INTERFACE ITF_Device EXTENDS ITF_BASE

PROPERTY Homed : BOOL
GET
END_GET
SET
END_SET
END_PROPERTY

METHOD mAbort : E_CmdState
VAR_INPUT
	I_bExecute : BOOL;
END_VAR
END_METHOD

METHOD mAutomatic : E_CmdState
VAR_INPUT
	I_bExecute : BOOL;
END_VAR
END_METHOD

METHOD mDone : E_CmdState
VAR_INPUT
END_VAR
END_METHOD

METHOD mHold : E_CmdState
VAR_INPUT
	I_bExecute : BOOL;
END_VAR
END_METHOD

METHOD mHome : E_CmdState
VAR_INPUT
	I_bExecute : BOOL;
END_VAR
END_METHOD

PROPERTY Mode : E_Mode
GET
END_GET
SET
END_SET
END_PROPERTY

METHOD mRelease : E_CmdState
VAR_INPUT
	I_bExecute : BOOL;
END_VAR
END_METHOD

METHOD mSequence : E_CmdState
VAR_INPUT
	I_bExecute : BOOL;
END_VAR
END_METHOD

METHOD mService : E_CmdState
VAR_INPUT
	I_bExecute : BOOL;
END_VAR
END_METHOD

METHOD mStop : E_CmdState
VAR_INPUT
	I_bExecute : BOOL;
END_VAR
END_METHOD

PROPERTY Ready : BOOL
GET
END_GET
SET
END_SET
END_PROPERTY

PROPERTY SequenceBusy : BOOL
GET
END_GET
SET
END_SET
END_PROPERTY

PROPERTY SequenceDone : BOOL
GET
END_GET
SET
END_SET
END_PROPERTY

END_INTERFACE

(* stored: Version 1.1.0.1, ProductVersion 3.1.4026.18
   Itf ITF_Device: Id {7c7c0ada-9da2-4ea4-a6eb-5bdbbf502dd6}
   Folder 01 Properties: Id {cc599803-8df0-4524-b56e-e6f8332deeb0}
   Folder 02 Methode: Id {8d03e7f7-1295-4a10-8500-54223f6c93df}
   Property Homed: Id {e0b0dbb4-f26b-41da-9728-17a21e3e50b5}
   Get Get: Id {b29716a5-bb80-4dae-9f4b-48cd3af13c02}
   Set Set: Id {c173668d-1e20-490e-b2a6-a314d734dc62}
   Method mAbort: Id {c49357ee-7419-4b69-b3cb-4341d2ee13d7}
   Method mAutomatic: Id {2d6cc853-f349-4892-b830-c8d902fec512}
   Method mDone: Id {ab0168ac-f476-4285-a122-68c9646e188c}
   Method mHold: Id {731bcd95-814c-4609-aa5e-a6712b35be37}
   Method mHome: Id {8c5e9607-f090-4f86-b53e-de4094b3fc51}
   Property Mode: Id {b4148d7b-1cf4-4690-8b11-f60ccf8fdb97}
   Get Get: Id {1764c7ca-5320-4c72-952b-b11de84e4a86}
   Set Set: Id {84b839d5-3e71-4766-9ef6-014419011dfe}
   Method mRelease: Id {39840917-54ed-488a-8e37-97e1ca73b28a}
   Method mSequence: Id {2de450d3-e14b-44df-ad83-42812f65ff1e}
   Method mService: Id {77e7e75c-3f71-4063-a921-5cc7e456b4a1}
   Method mStop: Id {dcef2cbd-175d-4efc-8e1c-1281a72f37b3}
   Property Ready: Id {47c16123-6529-4896-a7e2-12f8732a490d}
   Get Get: Id {0ffcaf96-efe5-4f3a-a02e-5895995aeb20}
   Set Set: Id {7f9ce145-10dd-4e65-9e06-ac93546155b2}
   Property SequenceBusy: Id {a4aff21a-c0f2-4f16-8fee-4bfeaa2eeabc}
   Get Get: Id {735e9e3b-26a3-49a1-87bb-52339686aefb}
   Set Set: Id {9efefb20-aa7d-4888-9b6a-1af16aefafce}
   Property SequenceDone: Id {f90f25ed-37ea-4ee3-b087-933acca26089}
   Get Get: Id {b6b79f53-27e7-470b-b01a-f1b7e039cb36}
   Set Set: Id {44443755-5c67-45ab-b267-791801d9ad44} *)
